// TIA Portal V19 export
VAR_GLOBAL   // PLC tag table "DemoCase"
   PB_Green_1200 AT %I0.0 : Bool;
   PB_Green_Lamp_1200 AT %Q0.0 : Bool;
   PB_Blue_1200 AT %I0.1 : Bool;
   PB_Blue_Lamp_1200 AT %Q0.1 : Bool;
   TopLights_Green_1200 AT %Q0.5 : Bool;
   TopLights_Red_1200 AT %Q0.6 : Bool;
   TopLights_Blue_1200 AT %Q0.7 : Bool;
   POT3_Upper_1200 AT %IW64 : Int;
   DataFrom1500 AT %IW4 : Word;
   IDevice AT %IB4 : Byte;
END_VAR
